PROGRAM MAIN
VAR
	
	x : BOOL;

END_VAR

;

END_PROGRAM

(* stored: Version 1.1.0.1, ProductVersion 3.1.4024.3
   POU MAIN: Id {2c804c71-a82c-4ec0-9b03-1208cfeebb79}, SpecialFunc None *)
